FUNCTION_BLOCK FB_HasInstanceNameImpl EXTENDS FB_HasInstanceName
VAR_INPUT
END_VAR
VAR_OUTPUT
END_VAR
VAR
END_VAR

END_FUNCTION_BLOCK

(* stored: Version 1.1.0.1, ProductVersion 3.1.4024.13
   POU FB_HasInstanceNameImpl: Id {1f529c36-7d92-0d2d-3534-c61eede3bd33}, SpecialFunc None *)
